# EPICS IOC start-up script: iocsh/computer-3p.iocsh
#
#   iocshLoad("$(superv_DIR)/computer-3p.iocsh")

#- ###                superv    iocsh               ###
#- ####################################################
#- >> Mandatory
#- IP_ADDR - IP address of the host
#- P	   - PV Prefix
#- PART1   - name of the first partition
#- PART2   - name of the first partition
#- PART3   - name of the first partition
#-
#- >> Optional
#- CH1     - SNMP variable channel (default 1)
#- CH2     - SNMP variable channel (default 2)
#- CH3     - SNMP variable channel (default 3)

devSnmpSetSnmpVersion($(IP_ADDR),SNMP_VERSION_2c)
dbLoadRecords("diskTable.template","P=$(P),PART=$(PART1),PASSWD=freia_secret,H=$(IP_ADDR),CHAN=$(CH1=1),HI=85,HH=95")
dbLoadRecords("diskTable.template","P=$(P),PART=$(PART2),PASSWD=freia_secret,H=$(IP_ADDR),CHAN=$(CH2=2),HI=85,HH=95")
dbLoadRecords("diskTable.template","P=$(P),PART=$(PART3),PASSWD=freia_secret,H=$(IP_ADDR),CHAN=$(CH3=3),HI=85,HH=95")
dbLoadRecords("hostSuperv.template","P=$(P),PASSWD=freia_secret,H=$(IP_ADDR)")
